// TIA Portal V15.1 export
// export: Created 2024-05-17T05:38:57.0702685Z, ExportSetting WithDefaults, DisplayName Totally Integrated Automation Portal, DisplayVersion V15.1 Update 5, DisplayName TIA Portal Openness, DisplayVersion V15.1 Update 5, DisplayName SINAMICS Startdrive Advanced, DisplayVersion V15.1, DisplayName G130, G150, S120, S150, SINAMICS MV, S210, DisplayVersion V15.1, DisplayName G110M, G120, G120C, G120D, G120P, DisplayVersion V15.1, DisplayName STEP 7 Professional, DisplayVersion V15.1 Update 5, DisplayName STEP 7 Safety, DisplayVersion V15.1, DisplayName WinCC Professional, DisplayVersion V15.1 Update 5, DisplayName SIMATIC Visualization Architect, DisplayVersion V15.1
FUNCTION "209210ZS01AEAK" : Void   // FC321, FBD
TITLE = 209210ZS01AEAK
{ S7_Optimized_Access := 'TRUE' }
AUTHOR : VCC
VERSION : 0.1
// stored: AutoNumber false, IsIECCheckEnabled false, SetENOAutomatically False, UDAEnableTagReadback false
   VAR_OUTPUT
      O_AlarmA : Bool;   // Alarm A
      O_AlarmB : Bool;   // Alarm B
      O_AlarmC : Bool;   // Alarm C
      O_AlarmD : Bool;   // Alarm D
      O_AlarmABCondition : Bool;   // Alarm AB condition
      H_IAnim : Word;   // For animation of icon
   END_VAR
BEGIN

REGION Network 1: **** --------------------- AE01 --------------------- ****
END_REGION

REGION Network 2: **** 2.2 Alarms - Alarm generation **** AE01E3FS07 // CH1 - 24VDC Fuse - ModeZone210 - Switch / Busnode 210AX01 & 210AS10
   // 24VDC Fuse - ModeZone210 - Switch / Busnode 210AX01 & 210AS10
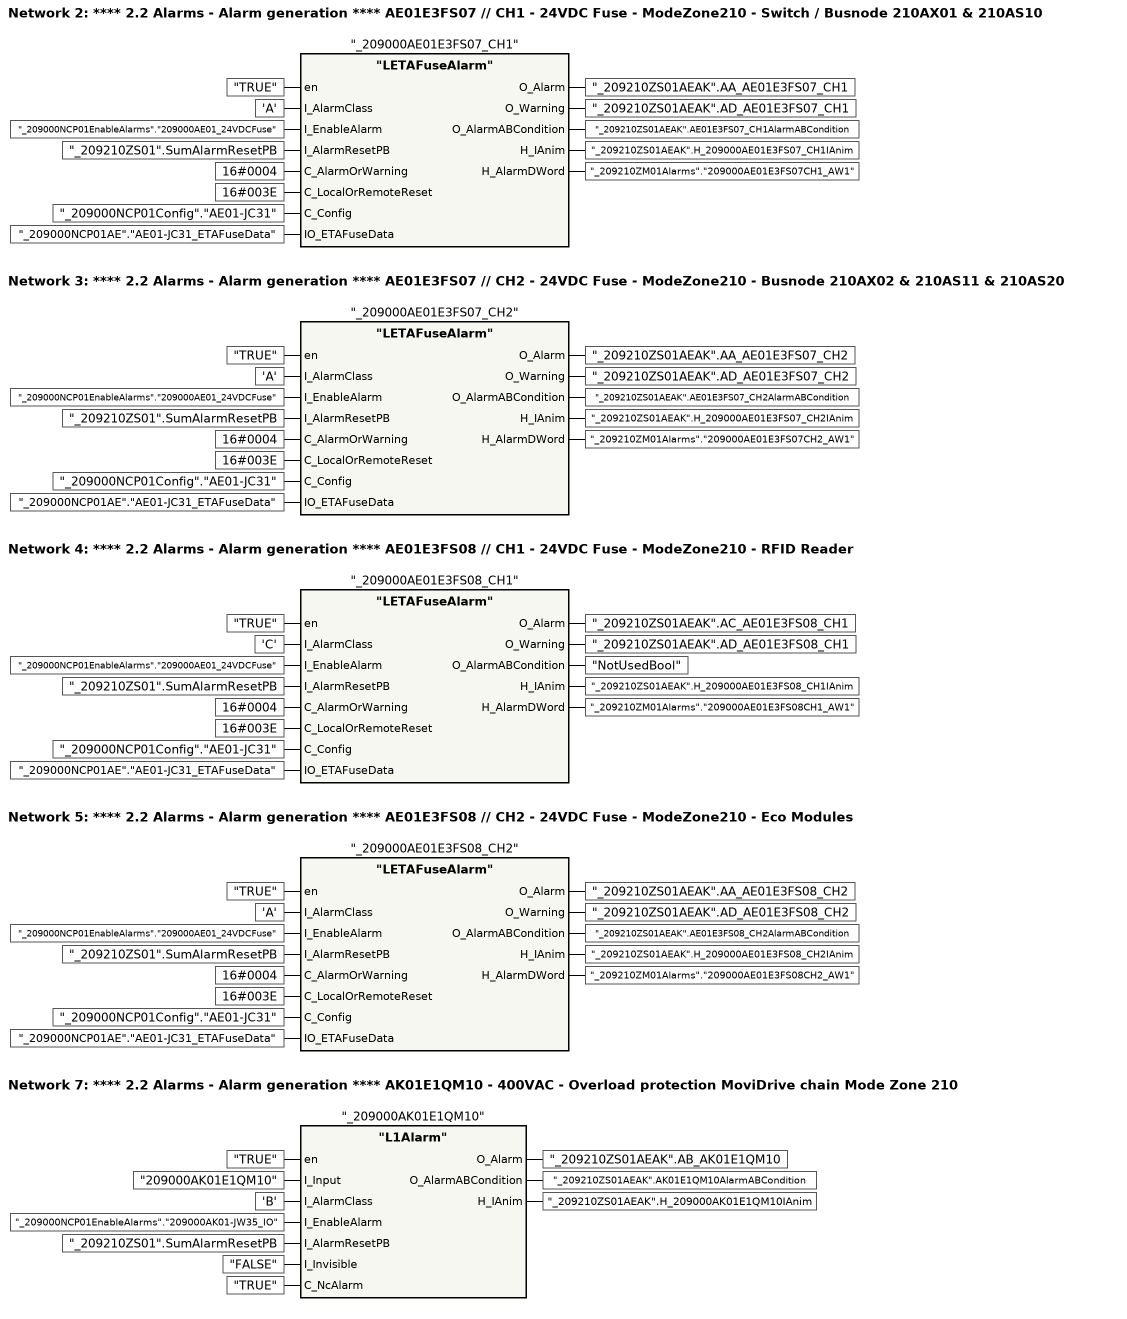
   IF "TRUE" THEN
       "_209000AE01E3FS07_CH1"(I_AlarmClass := 'A',   // "LETAFuseAlarm"
                               I_EnableAlarm := "_209000NCP01EnableAlarms"."209000AE01_24VDCFuse",
                               I_AlarmResetPB := "_209210ZS01".SumAlarmResetPB,
                               C_AlarmOrWarning := 16#0004,
                               C_LocalOrRemoteReset := 16#003E,
                               C_Config := "_209000NCP01Config"."AE01-JC31",
                               IO_ETAFuseData := "_209000NCP01AE"."AE01-JC31_ETAFuseData",
                               O_Alarm => "_209210ZS01AEAK".AA_AE01E3FS07_CH1,
                               O_Warning => "_209210ZS01AEAK".AD_AE01E3FS07_CH1,
                               O_AlarmABCondition => "_209210ZS01AEAK".AE01E3FS07_CH1AlarmABCondition,
                               H_IAnim => "_209210ZS01AEAK".H_209000AE01E3FS07_CH1IAnim,
                               H_AlarmDWord => "_209210ZM01Alarms"."209000AE01E3FS07CH1_AW1");
   END_IF;
END_REGION

REGION Network 3: **** 2.2 Alarms - Alarm generation **** AE01E3FS07 // CH2 - 24VDC Fuse - ModeZone210 - Busnode 210AX02 & 210AS11 & 210AS20
   // 24VDC Fuse - ModeZone210 - Busnode 210AX02 & 210AS11 & 210AS20
   IF "TRUE" THEN
       "_209000AE01E3FS07_CH2"(I_AlarmClass := 'A',   // "LETAFuseAlarm"
                               I_EnableAlarm := "_209000NCP01EnableAlarms"."209000AE01_24VDCFuse",
                               I_AlarmResetPB := "_209210ZS01".SumAlarmResetPB,
                               C_AlarmOrWarning := 16#0004,
                               C_LocalOrRemoteReset := 16#003E,
                               C_Config := "_209000NCP01Config"."AE01-JC31",
                               IO_ETAFuseData := "_209000NCP01AE"."AE01-JC31_ETAFuseData",
                               O_Alarm => "_209210ZS01AEAK".AA_AE01E3FS07_CH2,
                               O_Warning => "_209210ZS01AEAK".AD_AE01E3FS07_CH2,
                               O_AlarmABCondition => "_209210ZS01AEAK".AE01E3FS07_CH2AlarmABCondition,
                               H_IAnim => "_209210ZS01AEAK".H_209000AE01E3FS07_CH2IAnim,
                               H_AlarmDWord => "_209210ZM01Alarms"."209000AE01E3FS07CH2_AW1");
   END_IF;
END_REGION

REGION Network 4: **** 2.2 Alarms - Alarm generation **** AE01E3FS08 // CH1 - 24VDC Fuse - ModeZone210 - RFID Reader
   // 24VDC Fuse - ModeZone210 - RFID Reader
   IF "TRUE" THEN
       "_209000AE01E3FS08_CH1"(I_AlarmClass := 'C',   // "LETAFuseAlarm"
                               I_EnableAlarm := "_209000NCP01EnableAlarms"."209000AE01_24VDCFuse",
                               I_AlarmResetPB := "_209210ZS01".SumAlarmResetPB,
                               C_AlarmOrWarning := 16#0004,
                               C_LocalOrRemoteReset := 16#003E,
                               C_Config := "_209000NCP01Config"."AE01-JC31",
                               IO_ETAFuseData := "_209000NCP01AE"."AE01-JC31_ETAFuseData",
                               O_Alarm => "_209210ZS01AEAK".AC_AE01E3FS08_CH1,
                               O_Warning => "_209210ZS01AEAK".AD_AE01E3FS08_CH1,
                               O_AlarmABCondition => "NotUsedBool",
                               H_IAnim => "_209210ZS01AEAK".H_209000AE01E3FS08_CH1IAnim,
                               H_AlarmDWord => "_209210ZM01Alarms"."209000AE01E3FS08CH1_AW1");
   END_IF;
END_REGION

REGION Network 5: **** 2.2 Alarms - Alarm generation **** AE01E3FS08 // CH2 - 24VDC Fuse - ModeZone210 - Eco Modules
   // 24VDC Fuse - ModeZone210 - Eco Modules
   IF "TRUE" THEN
       "_209000AE01E3FS08_CH2"(I_AlarmClass := 'A',   // "LETAFuseAlarm"
                               I_EnableAlarm := "_209000NCP01EnableAlarms"."209000AE01_24VDCFuse",
                               I_AlarmResetPB := "_209210ZS01".SumAlarmResetPB,
                               C_AlarmOrWarning := 16#0004,
                               C_LocalOrRemoteReset := 16#003E,
                               C_Config := "_209000NCP01Config"."AE01-JC31",
                               IO_ETAFuseData := "_209000NCP01AE"."AE01-JC31_ETAFuseData",
                               O_Alarm => "_209210ZS01AEAK".AA_AE01E3FS08_CH2,
                               O_Warning => "_209210ZS01AEAK".AD_AE01E3FS08_CH2,
                               O_AlarmABCondition => "_209210ZS01AEAK".AE01E3FS08_CH2AlarmABCondition,
                               H_IAnim => "_209210ZS01AEAK".H_209000AE01E3FS08_CH2IAnim,
                               H_AlarmDWord => "_209210ZM01Alarms"."209000AE01E3FS08CH2_AW1");
   END_IF;
END_REGION

REGION Network 6: **** --------------------- AK01 --------------------- ****
END_REGION

REGION Network 7: **** 2.2 Alarms - Alarm generation **** AK01E1QM10 - 400VAC - Overload protection MoviDrive chain Mode Zone 210
   // 400VAC - Overload protection MoviDrive chain Mode Zone 210
   IF "TRUE" THEN
       "_209000AK01E1QM10"(I_Input := "209000AK01E1QM10",   // "L1Alarm"
                           I_AlarmClass := 'B',
                           I_EnableAlarm := "_209000NCP01EnableAlarms"."209000AK01-JW35_IO",
                           I_AlarmResetPB := "_209210ZS01".SumAlarmResetPB,
                           I_Invisible := "FALSE",
                           C_NcAlarm := "TRUE",
                           O_Alarm => "_209210ZS01AEAK".AB_AK01E1QM10,
                           O_AlarmABCondition => "_209210ZS01AEAK".AK01E1QM10AlarmABCondition,
                           H_IAnim => "_209210ZS01AEAK".H_209000AK01E1QM10IAnim);
   END_IF;
END_REGION

REGION Network 8: **** 2.2 Alarms - Alarm generation **** AK01E1QM11 - 400VAC - Overload protection MoviFit chain Mode Zone 210
   // 400VAC - Overload protection MoviFit chain Mode Zone 210
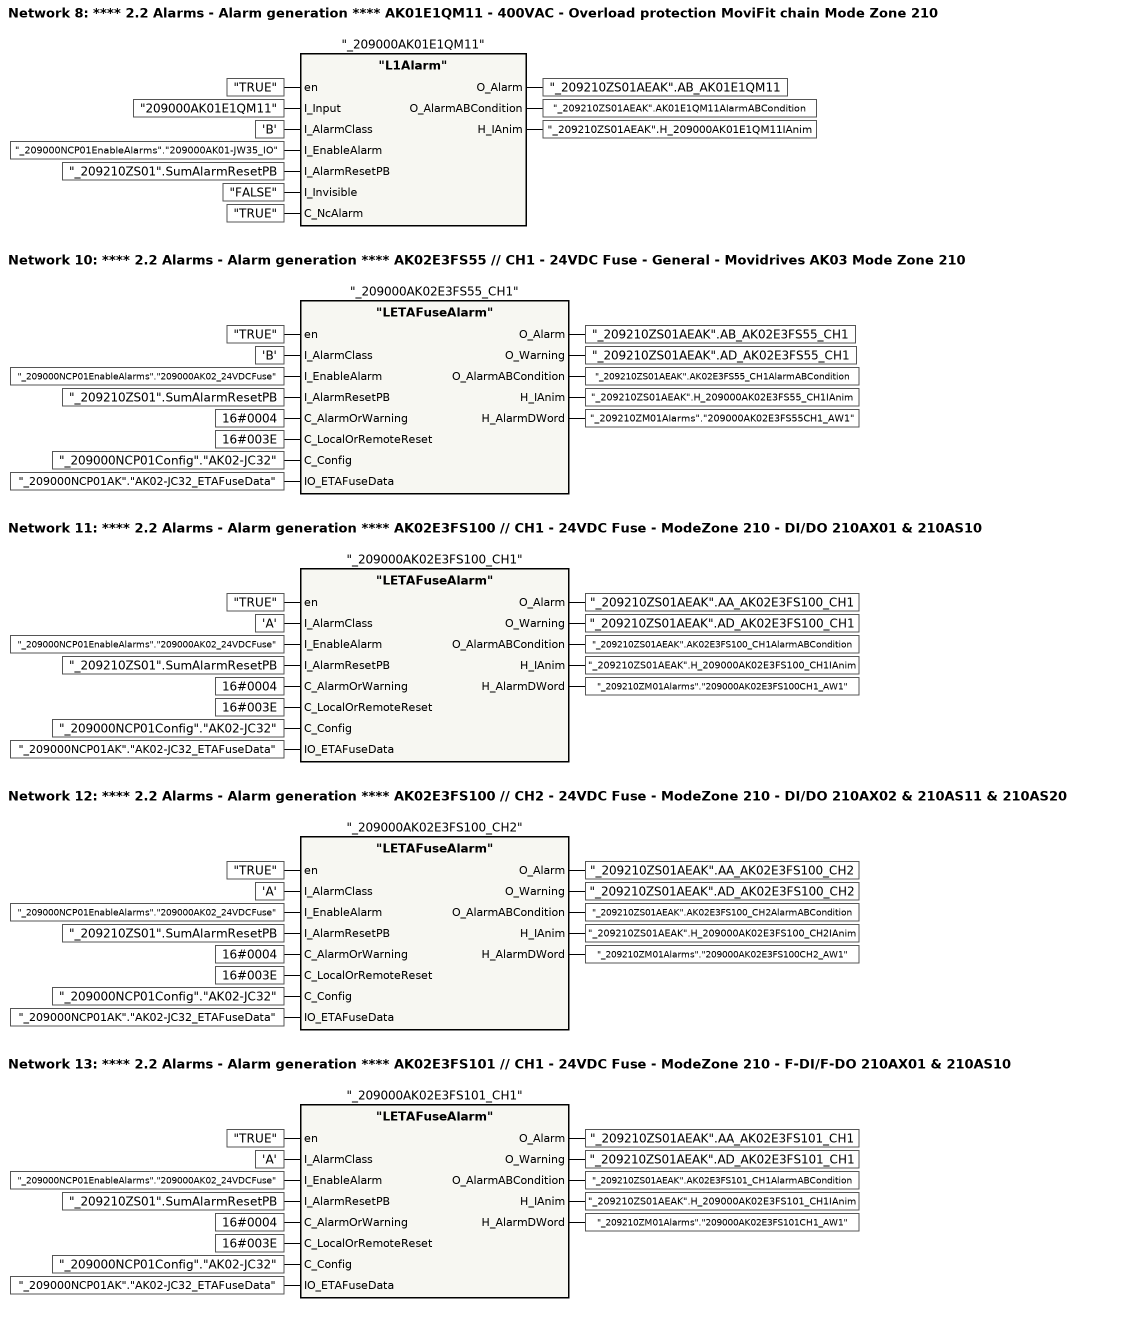
   IF "TRUE" THEN
       "_209000AK01E1QM11"(I_Input := "209000AK01E1QM11",   // "L1Alarm"
                           I_AlarmClass := 'B',
                           I_EnableAlarm := "_209000NCP01EnableAlarms"."209000AK01-JW35_IO",
                           I_AlarmResetPB := "_209210ZS01".SumAlarmResetPB,
                           I_Invisible := "FALSE",
                           C_NcAlarm := "TRUE",
                           O_Alarm => "_209210ZS01AEAK".AB_AK01E1QM11,
                           O_AlarmABCondition => "_209210ZS01AEAK".AK01E1QM11AlarmABCondition,
                           H_IAnim => "_209210ZS01AEAK".H_209000AK01E1QM11IAnim);
   END_IF;
END_REGION

REGION Network 9: **** --------------------- AK02 --------------------- ****
END_REGION

REGION Network 10: **** 2.2 Alarms - Alarm generation **** AK02E3FS55 // CH1 - 24VDC Fuse - General - Movidrives AK03 Mode Zone 210
   // 24VDC Fuse - General - Movidrives AK03 Mode Zone 210
   IF "TRUE" THEN
       "_209000AK02E3FS55_CH1"(I_AlarmClass := 'B',   // "LETAFuseAlarm"
                               I_EnableAlarm := "_209000NCP01EnableAlarms"."209000AK02_24VDCFuse",
                               I_AlarmResetPB := "_209210ZS01".SumAlarmResetPB,
                               C_AlarmOrWarning := 16#0004,
                               C_LocalOrRemoteReset := 16#003E,
                               C_Config := "_209000NCP01Config"."AK02-JC32",
                               IO_ETAFuseData := "_209000NCP01AK"."AK02-JC32_ETAFuseData",
                               O_Alarm => "_209210ZS01AEAK".AB_AK02E3FS55_CH1,
                               O_Warning => "_209210ZS01AEAK".AD_AK02E3FS55_CH1,
                               O_AlarmABCondition => "_209210ZS01AEAK".AK02E3FS55_CH1AlarmABCondition,
                               H_IAnim => "_209210ZS01AEAK".H_209000AK02E3FS55_CH1IAnim,
                               H_AlarmDWord => "_209210ZM01Alarms"."209000AK02E3FS55CH1_AW1");
   END_IF;
END_REGION

REGION Network 11: **** 2.2 Alarms - Alarm generation **** AK02E3FS100 // CH1 - 24VDC Fuse - ModeZone 210 - DI/DO 210AX01 & 210AS10
   // 24VDC Fuse - ModeZone 210 - DI/DO 210AX01 & 210AS10
   IF "TRUE" THEN
       "_209000AK02E3FS100_CH1"(I_AlarmClass := 'A',   // "LETAFuseAlarm"
                               I_EnableAlarm := "_209000NCP01EnableAlarms"."209000AK02_24VDCFuse",
                               I_AlarmResetPB := "_209210ZS01".SumAlarmResetPB,
                               C_AlarmOrWarning := 16#0004,
                               C_LocalOrRemoteReset := 16#003E,
                               C_Config := "_209000NCP01Config"."AK02-JC32",
                               IO_ETAFuseData := "_209000NCP01AK"."AK02-JC32_ETAFuseData",
                               O_Alarm => "_209210ZS01AEAK".AA_AK02E3FS100_CH1,
                               O_Warning => "_209210ZS01AEAK".AD_AK02E3FS100_CH1,
                               O_AlarmABCondition => "_209210ZS01AEAK".AK02E3FS100_CH1AlarmABCondition,
                               H_IAnim => "_209210ZS01AEAK".H_209000AK02E3FS100_CH1IAnim,
                               H_AlarmDWord => "_209210ZM01Alarms"."209000AK02E3FS100CH1_AW1");
   END_IF;
END_REGION

REGION Network 12: **** 2.2 Alarms - Alarm generation **** AK02E3FS100 // CH2 - 24VDC Fuse - ModeZone 210 - DI/DO 210AX02 & 210AS11 & 210AS20
   // 24VDC Fuse - ModeZone 210 - DI/DO 210AX02 & 210AS11 & 210AS20
   IF "TRUE" THEN
       "_209000AK02E3FS100_CH2"(I_AlarmClass := 'A',   // "LETAFuseAlarm"
                               I_EnableAlarm := "_209000NCP01EnableAlarms"."209000AK02_24VDCFuse",
                               I_AlarmResetPB := "_209210ZS01".SumAlarmResetPB,
                               C_AlarmOrWarning := 16#0004,
                               C_LocalOrRemoteReset := 16#003E,
                               C_Config := "_209000NCP01Config"."AK02-JC32",
                               IO_ETAFuseData := "_209000NCP01AK"."AK02-JC32_ETAFuseData",
                               O_Alarm => "_209210ZS01AEAK".AA_AK02E3FS100_CH2,
                               O_Warning => "_209210ZS01AEAK".AD_AK02E3FS100_CH2,
                               O_AlarmABCondition => "_209210ZS01AEAK".AK02E3FS100_CH2AlarmABCondition,
                               H_IAnim => "_209210ZS01AEAK".H_209000AK02E3FS100_CH2IAnim,
                               H_AlarmDWord => "_209210ZM01Alarms"."209000AK02E3FS100CH2_AW1");
   END_IF;
END_REGION

REGION Network 13: **** 2.2 Alarms - Alarm generation **** AK02E3FS101 // CH1 - 24VDC Fuse - ModeZone 210 - F-DI/F-DO 210AX01 & 210AS10
   // 24VDC Fuse - ModeZone 210 - F-DI/F-DO 210AX01 & 210AS10
   IF "TRUE" THEN
       "_209000AK02E3FS101_CH1"(I_AlarmClass := 'A',   // "LETAFuseAlarm"
                               I_EnableAlarm := "_209000NCP01EnableAlarms"."209000AK02_24VDCFuse",
                               I_AlarmResetPB := "_209210ZS01".SumAlarmResetPB,
                               C_AlarmOrWarning := 16#0004,
                               C_LocalOrRemoteReset := 16#003E,
                               C_Config := "_209000NCP01Config"."AK02-JC32",
                               IO_ETAFuseData := "_209000NCP01AK"."AK02-JC32_ETAFuseData",
                               O_Alarm => "_209210ZS01AEAK".AA_AK02E3FS101_CH1,
                               O_Warning => "_209210ZS01AEAK".AD_AK02E3FS101_CH1,
                               O_AlarmABCondition => "_209210ZS01AEAK".AK02E3FS101_CH1AlarmABCondition,
                               H_IAnim => "_209210ZS01AEAK".H_209000AK02E3FS101_CH1IAnim,
                               H_AlarmDWord => "_209210ZM01Alarms"."209000AK02E3FS101CH1_AW1");
   END_IF;
END_REGION

REGION Network 14: **** 2.2 Alarms - Alarm generation **** AK02E3FS101 // CH2 - 24VDC Fuse - ModeZone 210 - F-DI/F-DO 210AX02 & 210AS11 & 210AS20
   // 24VDC Fuse - ModeZone 210 - F-DI/F-DO 210AX02 & 210AS11 & 210AS20
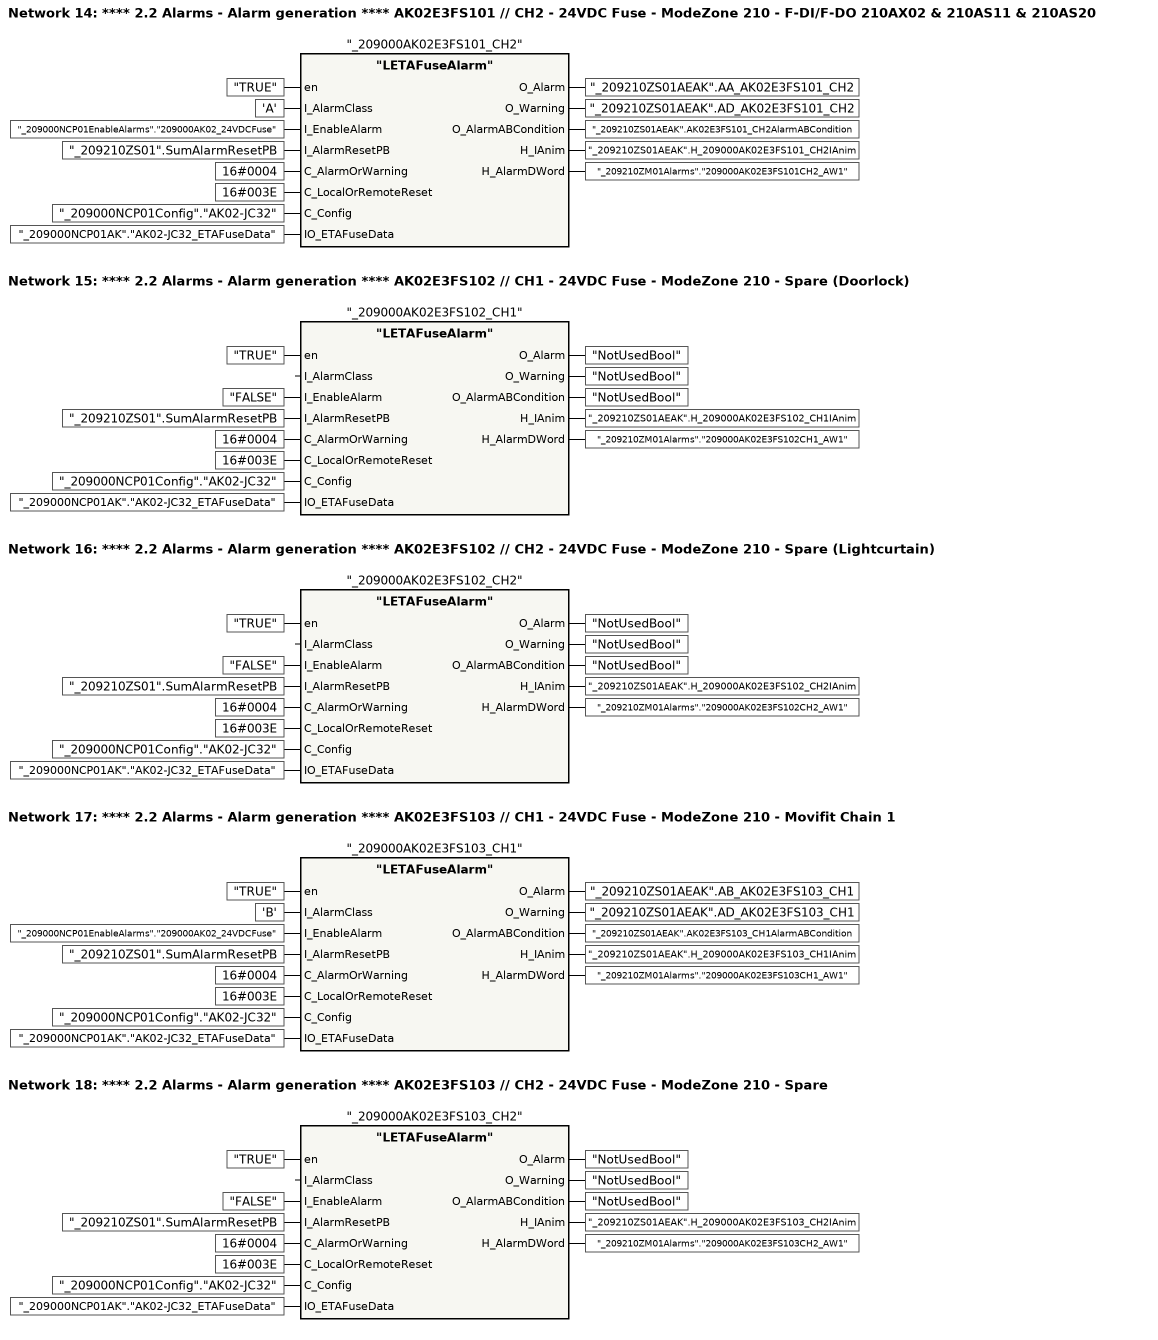
   IF "TRUE" THEN
       "_209000AK02E3FS101_CH2"(I_AlarmClass := 'A',   // "LETAFuseAlarm"
                               I_EnableAlarm := "_209000NCP01EnableAlarms"."209000AK02_24VDCFuse",
                               I_AlarmResetPB := "_209210ZS01".SumAlarmResetPB,
                               C_AlarmOrWarning := 16#0004,
                               C_LocalOrRemoteReset := 16#003E,
                               C_Config := "_209000NCP01Config"."AK02-JC32",
                               IO_ETAFuseData := "_209000NCP01AK"."AK02-JC32_ETAFuseData",
                               O_Alarm => "_209210ZS01AEAK".AA_AK02E3FS101_CH2,
                               O_Warning => "_209210ZS01AEAK".AD_AK02E3FS101_CH2,
                               O_AlarmABCondition => "_209210ZS01AEAK".AK02E3FS101_CH2AlarmABCondition,
                               H_IAnim => "_209210ZS01AEAK".H_209000AK02E3FS101_CH2IAnim,
                               H_AlarmDWord => "_209210ZM01Alarms"."209000AK02E3FS101CH2_AW1");
   END_IF;
END_REGION

REGION Network 15: **** 2.2 Alarms - Alarm generation **** AK02E3FS102 // CH1 - 24VDC Fuse - ModeZone 210 - Spare (Doorlock)
   // 24VDC Fuse - ModeZone 210 - Spare (Doorlock)
   IF "TRUE" THEN
       "_209000AK02E3FS102_CH1"(I_EnableAlarm := "FALSE",   // "LETAFuseAlarm"
                               I_AlarmResetPB := "_209210ZS01".SumAlarmResetPB,
                               C_AlarmOrWarning := 16#0004,
                               C_LocalOrRemoteReset := 16#003E,
                               C_Config := "_209000NCP01Config"."AK02-JC32",
                               IO_ETAFuseData := "_209000NCP01AK"."AK02-JC32_ETAFuseData",
                               O_Alarm => "NotUsedBool",
                               O_Warning => "NotUsedBool",
                               O_AlarmABCondition => "NotUsedBool",
                               H_IAnim => "_209210ZS01AEAK".H_209000AK02E3FS102_CH1IAnim,
                               H_AlarmDWord => "_209210ZM01Alarms"."209000AK02E3FS102CH1_AW1");
   END_IF;
END_REGION

REGION Network 16: **** 2.2 Alarms - Alarm generation **** AK02E3FS102 // CH2 - 24VDC Fuse - ModeZone 210 - Spare (Lightcurtain)
   // 24VDC Fuse - ModeZone 210 - Spare (Lightcurtain)
   IF "TRUE" THEN
       "_209000AK02E3FS102_CH2"(I_EnableAlarm := "FALSE",   // "LETAFuseAlarm"
                               I_AlarmResetPB := "_209210ZS01".SumAlarmResetPB,
                               C_AlarmOrWarning := 16#0004,
                               C_LocalOrRemoteReset := 16#003E,
                               C_Config := "_209000NCP01Config"."AK02-JC32",
                               IO_ETAFuseData := "_209000NCP01AK"."AK02-JC32_ETAFuseData",
                               O_Alarm => "NotUsedBool",
                               O_Warning => "NotUsedBool",
                               O_AlarmABCondition => "NotUsedBool",
                               H_IAnim => "_209210ZS01AEAK".H_209000AK02E3FS102_CH2IAnim,
                               H_AlarmDWord => "_209210ZM01Alarms"."209000AK02E3FS102CH2_AW1");
   END_IF;
END_REGION

REGION Network 17: **** 2.2 Alarms - Alarm generation **** AK02E3FS103 // CH1 - 24VDC Fuse - ModeZone 210 - Movifit Chain 1
   // 24VDC Fuse - ModeZone 210 - Movifit Chain 1
   IF "TRUE" THEN
       "_209000AK02E3FS103_CH1"(I_AlarmClass := 'B',   // "LETAFuseAlarm"
                               I_EnableAlarm := "_209000NCP01EnableAlarms"."209000AK02_24VDCFuse",
                               I_AlarmResetPB := "_209210ZS01".SumAlarmResetPB,
                               C_AlarmOrWarning := 16#0004,
                               C_LocalOrRemoteReset := 16#003E,
                               C_Config := "_209000NCP01Config"."AK02-JC32",
                               IO_ETAFuseData := "_209000NCP01AK"."AK02-JC32_ETAFuseData",
                               O_Alarm => "_209210ZS01AEAK".AB_AK02E3FS103_CH1,
                               O_Warning => "_209210ZS01AEAK".AD_AK02E3FS103_CH1,
                               O_AlarmABCondition => "_209210ZS01AEAK".AK02E3FS103_CH1AlarmABCondition,
                               H_IAnim => "_209210ZS01AEAK".H_209000AK02E3FS103_CH1IAnim,
                               H_AlarmDWord => "_209210ZM01Alarms"."209000AK02E3FS103CH1_AW1");
   END_IF;
END_REGION

REGION Network 18: **** 2.2 Alarms - Alarm generation **** AK02E3FS103 // CH2 - 24VDC Fuse - ModeZone 210 - Spare
   // 24VDC Fuse - ModeZone 210 - Spare
   IF "TRUE" THEN
       "_209000AK02E3FS103_CH2"(I_EnableAlarm := "FALSE",   // "LETAFuseAlarm"
                               I_AlarmResetPB := "_209210ZS01".SumAlarmResetPB,
                               C_AlarmOrWarning := 16#0004,
                               C_LocalOrRemoteReset := 16#003E,
                               C_Config := "_209000NCP01Config"."AK02-JC32",
                               IO_ETAFuseData := "_209000NCP01AK"."AK02-JC32_ETAFuseData",
                               O_Alarm => "NotUsedBool",
                               O_Warning => "NotUsedBool",
                               O_AlarmABCondition => "NotUsedBool",
                               H_IAnim => "_209210ZS01AEAK".H_209000AK02E3FS103_CH2IAnim,
                               H_AlarmDWord => "_209210ZM01Alarms"."209000AK02E3FS103CH2_AW1");
   END_IF;
END_REGION

REGION Network 19: **** --------------------- AK03 --------------------- ****
END_REGION

REGION Network 20: **** 2.2 Alarms - Alarm generation **** AK03E1QM130 - 400VAC - Overload protection Brake Resistor 209210CR21
   // 400VAC - Overload protection Brake Resistor 209210CR21
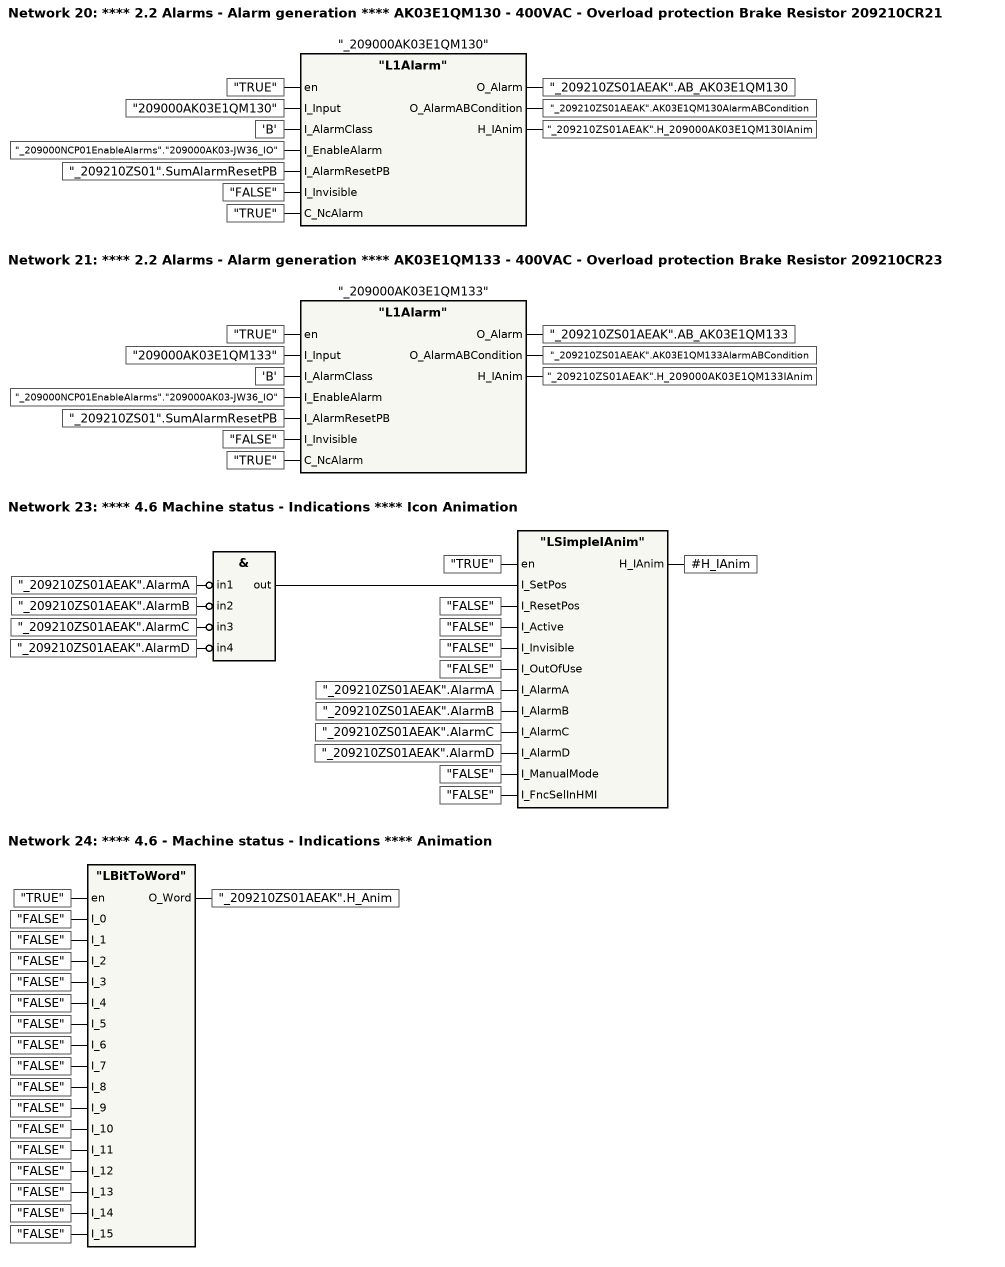
   IF "TRUE" THEN
       "_209000AK03E1QM130"(I_Input := "209000AK03E1QM130",   // "L1Alarm"
                            I_AlarmClass := 'B',
                            I_EnableAlarm := "_209000NCP01EnableAlarms"."209000AK03-JW36_IO",
                            I_AlarmResetPB := "_209210ZS01".SumAlarmResetPB,
                            I_Invisible := "FALSE",
                            C_NcAlarm := "TRUE",
                            O_Alarm => "_209210ZS01AEAK".AB_AK03E1QM130,
                            O_AlarmABCondition => "_209210ZS01AEAK".AK03E1QM130AlarmABCondition,
                            H_IAnim => "_209210ZS01AEAK".H_209000AK03E1QM130IAnim);
   END_IF;
END_REGION

REGION Network 21: **** 2.2 Alarms - Alarm generation **** AK03E1QM133 - 400VAC - Overload protection Brake Resistor 209210CR23
   // 400VAC - Overload protection Brake Resistor 209210CR23
   IF "TRUE" THEN
       "_209000AK03E1QM133"(I_Input := "209000AK03E1QM133",   // "L1Alarm"
                            I_AlarmClass := 'B',
                            I_EnableAlarm := "_209000NCP01EnableAlarms"."209000AK03-JW36_IO",
                            I_AlarmResetPB := "_209210ZS01".SumAlarmResetPB,
                            I_Invisible := "FALSE",
                            C_NcAlarm := "TRUE",
                            O_Alarm => "_209210ZS01AEAK".AB_AK03E1QM133,
                            O_AlarmABCondition => "_209210ZS01AEAK".AK03E1QM133AlarmABCondition,
                            H_IAnim => "_209210ZS01AEAK".H_209000AK03E1QM133IAnim);
   END_IF;
END_REGION

REGION Network 22: **** -------------------------------------------------- ****
END_REGION

REGION Network 23: **** 4.6 Machine status - Indications **** Icon Animation
   // Animation for icon
   IF "TRUE" THEN
       "LSimpleIAnim"(I_SetPos := NOT "_209210ZS01AEAK".AlarmA AND NOT "_209210ZS01AEAK".AlarmB AND NOT "_209210ZS01AEAK".AlarmC AND NOT "_209210ZS01AEAK".AlarmD,
                      I_ResetPos := "FALSE",
                      I_Active := "FALSE",
                      I_Invisible := "FALSE",
                      I_OutOfUse := "FALSE",
                      I_AlarmA := "_209210ZS01AEAK".AlarmA,
                      I_AlarmB := "_209210ZS01AEAK".AlarmB,
                      I_AlarmC := "_209210ZS01AEAK".AlarmC,
                      I_AlarmD := "_209210ZS01AEAK".AlarmD,
                      I_ManualMode := "FALSE",
                      I_FncSelInHMI := "FALSE",
                      H_IAnim => #H_IAnim);
   END_IF;
END_REGION

REGION Network 24: **** 4.6 - Machine status - Indications **** Animation
   // Animation
   IF "TRUE" THEN
       "LBitToWord"(I_0 := "FALSE",
                    I_1 := "FALSE",
                    I_2 := "FALSE",
                    I_3 := "FALSE",
                    I_4 := "FALSE",
                    I_5 := "FALSE",
                    I_6 := "FALSE",
                    I_7 := "FALSE",
                    I_8 := "FALSE",
                    I_9 := "FALSE",
                    I_10 := "FALSE",
                    I_11 := "FALSE",
                    I_12 := "FALSE",
                    I_13 := "FALSE",
                    I_14 := "FALSE",
                    I_15 := "FALSE",
                    O_Word => "_209210ZS01AEAK".H_Anim);
   END_IF;
END_REGION

NETWORK
TITLE = **** 4.6 - Machine Status - Indications **** Animation DB number
// DB number
      OPN   "_209210ZS01AEAK";
      L     DBNO;
      T     "_209210ZS01AEAK".H_DBnr;

REGION Network 26: **** 9 - Alarm Summary **** Alarm AB condition
   // Alarm AB condition
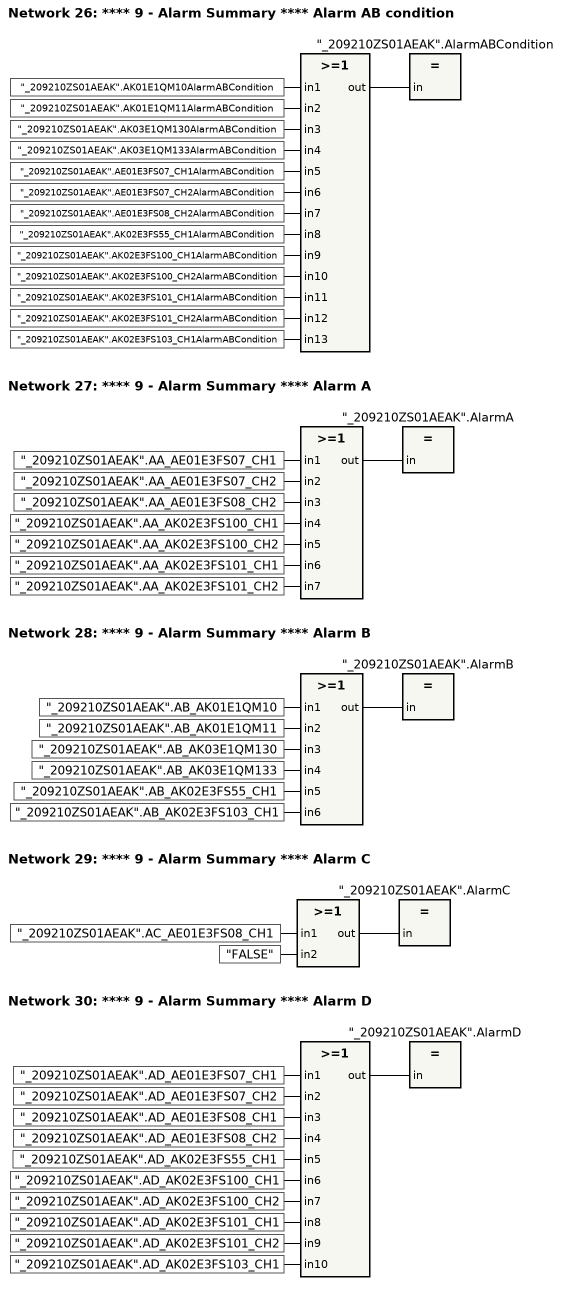
   "_209210ZS01AEAK".AlarmABCondition := "_209210ZS01AEAK".AK01E1QM10AlarmABCondition OR "_209210ZS01AEAK".AK01E1QM11AlarmABCondition OR "_209210ZS01AEAK".AK03E1QM130AlarmABCondition OR "_209210ZS01AEAK".AK03E1QM133AlarmABCondition OR "_209210ZS01AEAK".AE01E3FS07_CH1AlarmABCondition OR "_209210ZS01AEAK".AE01E3FS07_CH2AlarmABCondition OR "_209210ZS01AEAK".AE01E3FS08_CH2AlarmABCondition OR "_209210ZS01AEAK".AK02E3FS55_CH1AlarmABCondition OR "_209210ZS01AEAK".AK02E3FS100_CH1AlarmABCondition OR "_209210ZS01AEAK".AK02E3FS100_CH2AlarmABCondition OR "_209210ZS01AEAK".AK02E3FS101_CH1AlarmABCondition OR "_209210ZS01AEAK".AK02E3FS101_CH2AlarmABCondition OR "_209210ZS01AEAK".AK02E3FS103_CH1AlarmABCondition;
END_REGION

REGION Network 27: **** 9 - Alarm Summary **** Alarm A
   // Summary of alarms A
   "_209210ZS01AEAK".AlarmA := "_209210ZS01AEAK".AA_AE01E3FS07_CH1 OR "_209210ZS01AEAK".AA_AE01E3FS07_CH2 OR "_209210ZS01AEAK".AA_AE01E3FS08_CH2 OR "_209210ZS01AEAK".AA_AK02E3FS100_CH1 OR "_209210ZS01AEAK".AA_AK02E3FS100_CH2 OR "_209210ZS01AEAK".AA_AK02E3FS101_CH1 OR "_209210ZS01AEAK".AA_AK02E3FS101_CH2;
END_REGION

REGION Network 28: **** 9 - Alarm Summary **** Alarm B
   // Summary of alarms B
   "_209210ZS01AEAK".AlarmB := "_209210ZS01AEAK".AB_AK01E1QM10 OR "_209210ZS01AEAK".AB_AK01E1QM11 OR "_209210ZS01AEAK".AB_AK03E1QM130 OR "_209210ZS01AEAK".AB_AK03E1QM133 OR "_209210ZS01AEAK".AB_AK02E3FS55_CH1 OR "_209210ZS01AEAK".AB_AK02E3FS103_CH1;
END_REGION

REGION Network 29: **** 9 - Alarm Summary **** Alarm C
   // Summary of alarms C
   "_209210ZS01AEAK".AlarmC := "_209210ZS01AEAK".AC_AE01E3FS08_CH1 OR "FALSE";
END_REGION

REGION Network 30: **** 9 - Alarm Summary **** Alarm D
   // Summary of alarms D
   "_209210ZS01AEAK".AlarmD := "_209210ZS01AEAK".AD_AE01E3FS07_CH1 OR "_209210ZS01AEAK".AD_AE01E3FS07_CH2 OR "_209210ZS01AEAK".AD_AE01E3FS08_CH1 OR "_209210ZS01AEAK".AD_AE01E3FS08_CH2 OR "_209210ZS01AEAK".AD_AK02E3FS55_CH1 OR "_209210ZS01AEAK".AD_AK02E3FS100_CH1 OR "_209210ZS01AEAK".AD_AK02E3FS100_CH2 OR "_209210ZS01AEAK".AD_AK02E3FS101_CH1 OR "_209210ZS01AEAK".AD_AK02E3FS101_CH2 OR "_209210ZS01AEAK".AD_AK02E3FS103_CH1;
END_REGION

REGION Network 31: **** 9.1 - Alarm Output **** Alarm AB condition
   // Alarm AB condition
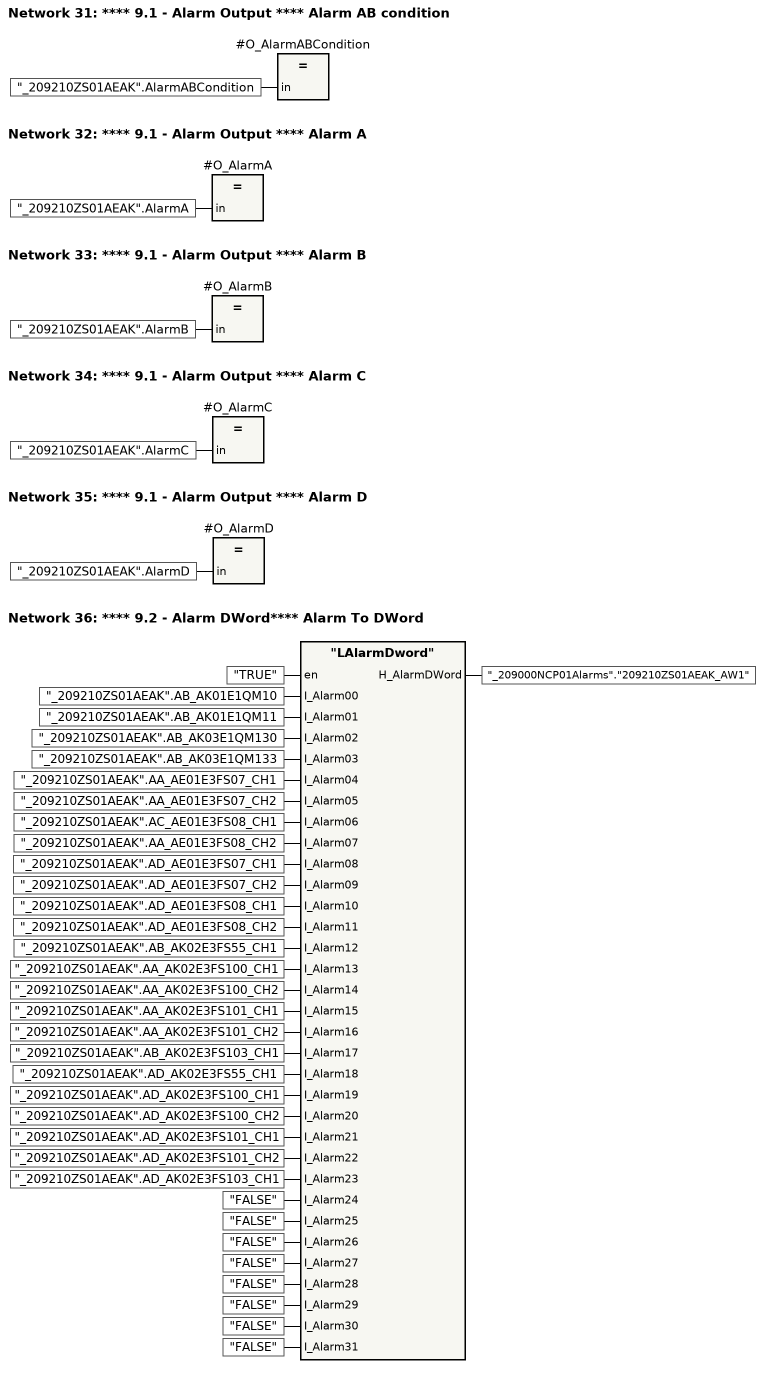
   #O_AlarmABCondition := "_209210ZS01AEAK".AlarmABCondition;
END_REGION

REGION Network 32: **** 9.1 - Alarm Output **** Alarm A
   // Summary of alarms A
   #O_AlarmA := "_209210ZS01AEAK".AlarmA;
END_REGION

REGION Network 33: **** 9.1 - Alarm Output **** Alarm B
   // Summary of alarms B
   #O_AlarmB := "_209210ZS01AEAK".AlarmB;
END_REGION

REGION Network 34: **** 9.1 - Alarm Output **** Alarm C
   // Summary of alarms C
   #O_AlarmC := "_209210ZS01AEAK".AlarmC;
END_REGION

REGION Network 35: **** 9.1 - Alarm Output **** Alarm D
   // Summary of alarms D
   #O_AlarmD := "_209210ZS01AEAK".AlarmD;
END_REGION

REGION Network 36: **** 9.2 - Alarm DWord**** Alarm To DWord
   // Alarm Word
   IF "TRUE" THEN
       "LAlarmDword"(I_Alarm00 := "_209210ZS01AEAK".AB_AK01E1QM10,
                     I_Alarm01 := "_209210ZS01AEAK".AB_AK01E1QM11,
                     I_Alarm02 := "_209210ZS01AEAK".AB_AK03E1QM130,
                     I_Alarm03 := "_209210ZS01AEAK".AB_AK03E1QM133,
                     I_Alarm04 := "_209210ZS01AEAK".AA_AE01E3FS07_CH1,
                     I_Alarm05 := "_209210ZS01AEAK".AA_AE01E3FS07_CH2,
                     I_Alarm06 := "_209210ZS01AEAK".AC_AE01E3FS08_CH1,
                     I_Alarm07 := "_209210ZS01AEAK".AA_AE01E3FS08_CH2,
                     I_Alarm08 := "_209210ZS01AEAK".AD_AE01E3FS07_CH1,
                     I_Alarm09 := "_209210ZS01AEAK".AD_AE01E3FS07_CH2,
                     I_Alarm10 := "_209210ZS01AEAK".AD_AE01E3FS08_CH1,
                     I_Alarm11 := "_209210ZS01AEAK".AD_AE01E3FS08_CH2,
                     I_Alarm12 := "_209210ZS01AEAK".AB_AK02E3FS55_CH1,
                     I_Alarm13 := "_209210ZS01AEAK".AA_AK02E3FS100_CH1,
                     I_Alarm14 := "_209210ZS01AEAK".AA_AK02E3FS100_CH2,
                     I_Alarm15 := "_209210ZS01AEAK".AA_AK02E3FS101_CH1,
                     I_Alarm16 := "_209210ZS01AEAK".AA_AK02E3FS101_CH2,
                     I_Alarm17 := "_209210ZS01AEAK".AB_AK02E3FS103_CH1,
                     I_Alarm18 := "_209210ZS01AEAK".AD_AK02E3FS55_CH1,
                     I_Alarm19 := "_209210ZS01AEAK".AD_AK02E3FS100_CH1,
                     I_Alarm20 := "_209210ZS01AEAK".AD_AK02E3FS100_CH2,
                     I_Alarm21 := "_209210ZS01AEAK".AD_AK02E3FS101_CH1,
                     I_Alarm22 := "_209210ZS01AEAK".AD_AK02E3FS101_CH2,
                     I_Alarm23 := "_209210ZS01AEAK".AD_AK02E3FS103_CH1,
                     I_Alarm24 := "FALSE",
                     I_Alarm25 := "FALSE",
                     I_Alarm26 := "FALSE",
                     I_Alarm27 := "FALSE",
                     I_Alarm28 := "FALSE",
                     I_Alarm29 := "FALSE",
                     I_Alarm30 := "FALSE",
                     I_Alarm31 := "FALSE",
                     H_AlarmDWord => "_209000NCP01Alarms"."209210ZS01AEAK_AW1");
   END_IF;
END_REGION
END_FUNCTION
